{attribute 'GeneratedUsingTerminal: EPP6228-0022-0016'}
{attribute addProperty BoxType "EPP6228-0022-0016"}
{attribute addProperty Id "State_Ch1AT %I*USINT1State_Ch2AT %I*USINT1State_Ch3AT %I*USINT1State_Ch4AT %I*USINT1State_Ch5AT %I*USINT1State_Ch6AT %I*USINT1State_Ch7AT %I*USINT1State_Ch8AT %I*USINT1"}
{attribute addProperty CRC "3341098441"}
{attribute addProperty Size "8"}
TYPE DeviceState_Inputs_C7251DC9 :
STRUCT
	{attribute addProperty Name "State_Ch1"}
	State_Ch1 AT %I* : USINT;
	{attribute addProperty Name "State_Ch2"}
	State_Ch2 AT %I* : USINT;
	{attribute addProperty Name "State_Ch3"}
	State_Ch3 AT %I* : USINT;
	{attribute addProperty Name "State_Ch4"}
	State_Ch4 AT %I* : USINT;
	{attribute addProperty Name "State_Ch5"}
	State_Ch5 AT %I* : USINT;
	{attribute addProperty Name "State_Ch6"}
	State_Ch6 AT %I* : USINT;
	{attribute addProperty Name "State_Ch7"}
	State_Ch7 AT %I* : USINT;
	{attribute addProperty Name "State_Ch8"}
	State_Ch8 AT %I* : USINT;
END_STRUCT
END_TYPE

(* stored: Version 1.2.0.0, ProductVersion 3.1.4024.9
   DUT DeviceState_Inputs_C7251DC9: Id {93d23277-1c01-49c6-9a96-7acaaec97367} *)
